(* Logix 5000 project; controller SX_V040001_C001 vendor 1 type 14 code 77 rev 16.23; software revision 16.04; part 3 of 35 *)
(* tags used below, declared in another part *)
   ALARM_BITS : INT[10];
   ALL_KINDS : INT[90];
   Basic : INT;
   G_DInput : DINT[3];
   G_DOutput : DINT[3];
   m_alarm_exist : BOOL;
   m_notstop : BOOL;
   METERING : INT[44];
   PARAMETER : INT[501];
   T_MET1_END : TIMER;
   T_MET2_END : TIMER;
   T_MET3_END : TIMER;
   T_MET4_END : TIMER;
   T_MET_VALVE_1 : TIMER;
   T_MET_VALVE_2 : TIMER;
   T_MET_VALVE_3 : TIMER;
   T_MET_VALVE_4 : TIMER;
   T_MET_VALVE_5 : TIMER;
   Z20 : COUNTER;
   Z21 : COUNTER;
   Z22 : COUNTER;
   Z23 : COUNTER;
   Z24 : COUNTER;
   Z25 : COUNTER;
   Z26 : COUNTER;
   Z27 : COUNTER;
   Z28 : COUNTER;
(* MainProgram, continued *)

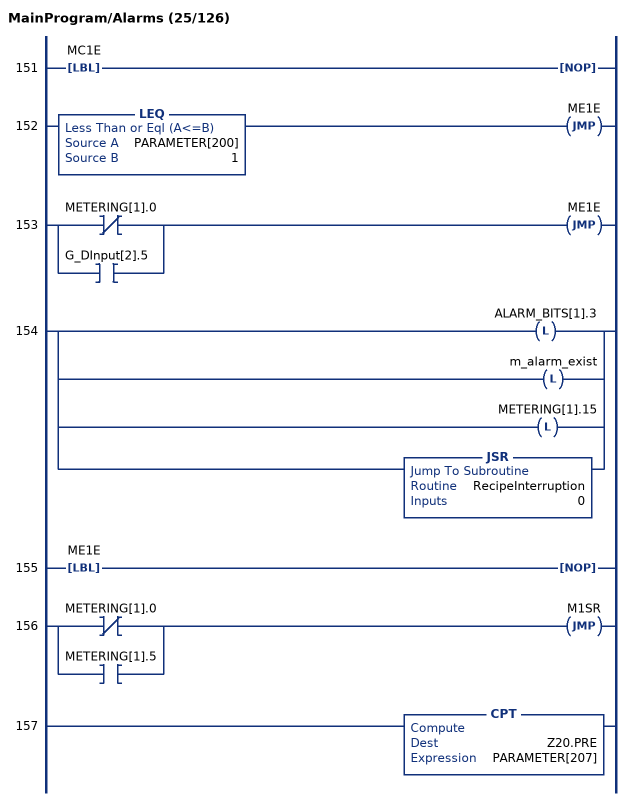
   [picture p46: MainProgram/Alarms rungs 151-157]
   151: LBL(MC1E)NOP();
   152: LEQ(PARAMETER[200],1)JMP(ME1E);
   153: [XIO(METERING[1].0) ,XIC(G_DInput[2].5) ]JMP(ME1E);
   154: [OTL(ALARM_BITS[1].3) ,OTL(m_alarm_exist) ,OTL(METERING[1].15) ,JSR(RecipeInterruption,0) ];
   155: LBL(ME1E)NOP();
   156: [XIO(METERING[1].0) ,XIC(METERING[1].5) ]JMP(M1SR);
   157: CPT(Z20.PRE,PARAMETER[207]);
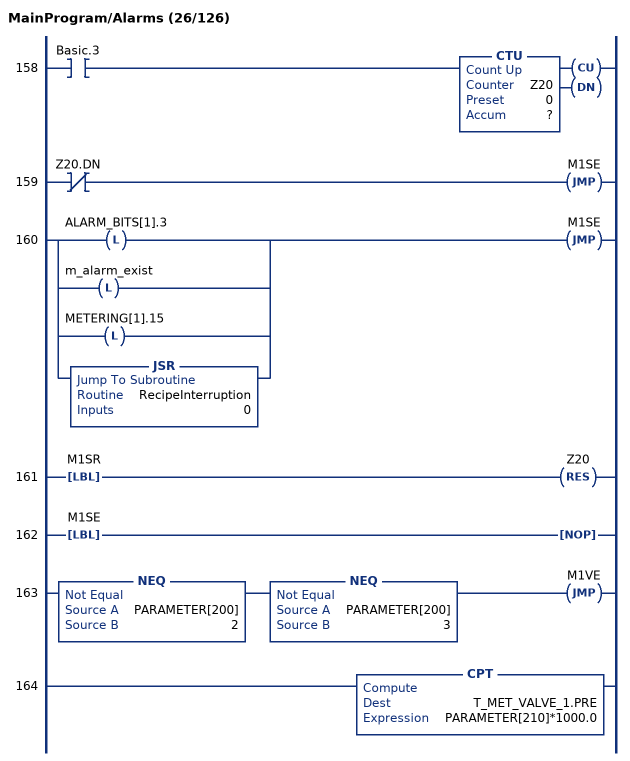
   158: XIC(Basic.3)CTU(Z20,?,?);
   159: XIO(Z20.DN)JMP(M1SE);
   160: [OTL(ALARM_BITS[1].3) ,OTL(m_alarm_exist) ,OTL(METERING[1].15) ,JSR(RecipeInterruption,0) ]JMP(M1SE);
   161: LBL(M1SR)RES(Z20);
   162: LBL(M1SE)NOP();
   163: NEQ(PARAMETER[200],2)NEQ(PARAMETER[200],3)JMP(M1VE);
   164: CPT(T_MET_VALVE_1.PRE,PARAMETER[210]*1000.0);
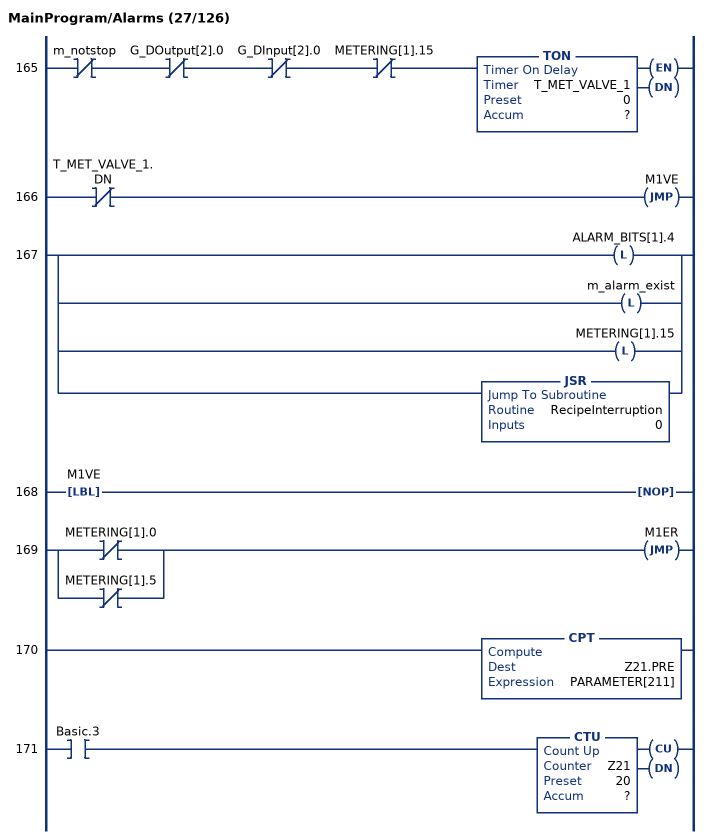
   165: XIO(m_notstop)XIO(G_DOutput[2].0)XIO(G_DInput[2].0)XIO(METERING[1].15)TON(T_MET_VALVE_1,?,?);
   166: XIO(T_MET_VALVE_1.DN)JMP(M1VE);
   167: [OTL(ALARM_BITS[1].4) ,OTL(m_alarm_exist) ,OTL(METERING[1].15) ,JSR(RecipeInterruption,0) ];
   168: LBL(M1VE)NOP();
   169: [XIO(METERING[1].0) ,XIO(METERING[1].5) ]JMP(M1ER);
   170: CPT(Z21.PRE,PARAMETER[211]);
   171: XIC(Basic.3)CTU(Z21,?,?);
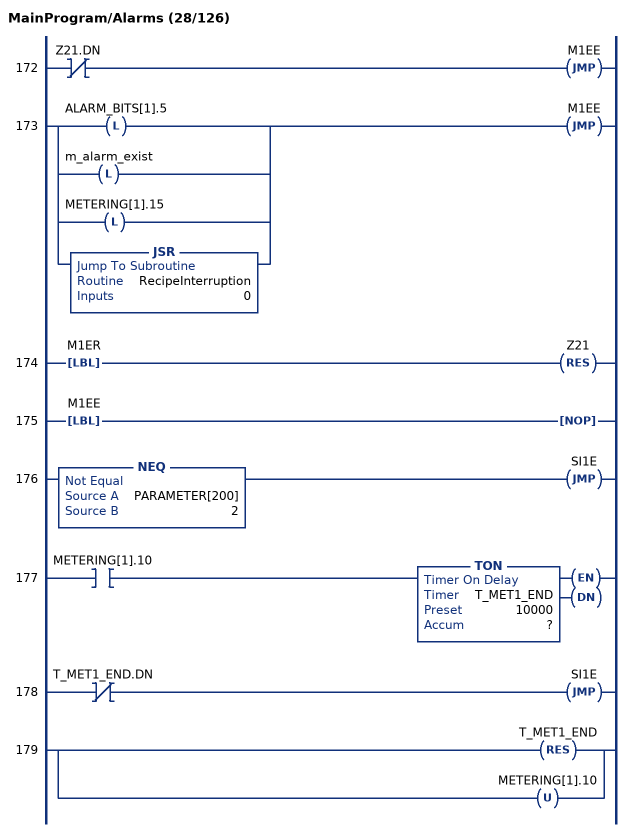
   172: XIO(Z21.DN)JMP(M1EE);
   173: [OTL(ALARM_BITS[1].5) ,OTL(m_alarm_exist) ,OTL(METERING[1].15) ,JSR(RecipeInterruption,0) ]JMP(M1EE);
   174: LBL(M1ER)RES(Z21);
   175: LBL(M1EE)NOP();
   176: NEQ(PARAMETER[200],2)JMP(SI1E);
   177: XIC(METERING[1].10)TON(T_MET1_END,?,?);
   178: XIO(T_MET1_END.DN)JMP(SI1E);
   179: [RES(T_MET1_END) ,OTU(METERING[1].10) ];
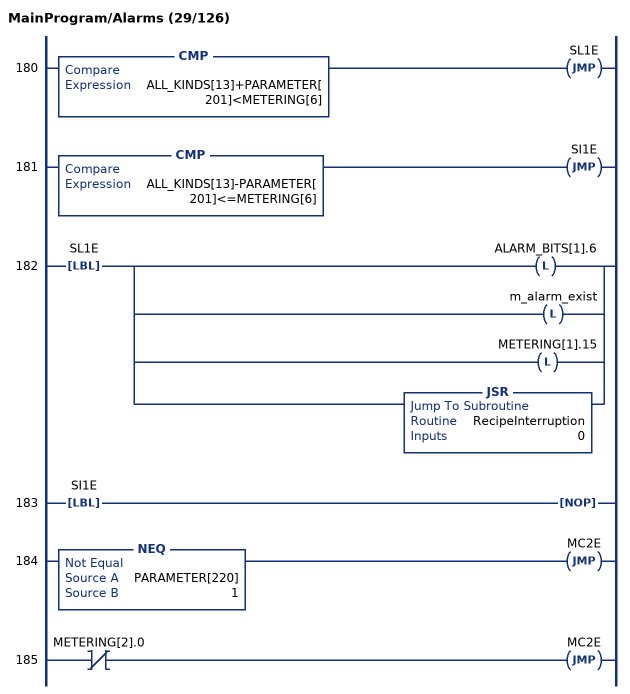
   180: CMP(ALL_KINDS[13]+PARAMETER[201]<METERING[6])JMP(SL1E);
   181: CMP(ALL_KINDS[13]-PARAMETER[201]<=METERING[6])JMP(SI1E);
   182: LBL(SL1E)[OTL(ALARM_BITS[1].6) ,OTL(m_alarm_exist) ,OTL(METERING[1].15) ,JSR(RecipeInterruption,0) ];
   183: LBL(SI1E)NOP();
   184: NEQ(PARAMETER[220],1)JMP(MC2E);
   185: XIO(METERING[2].0)JMP(MC2E);
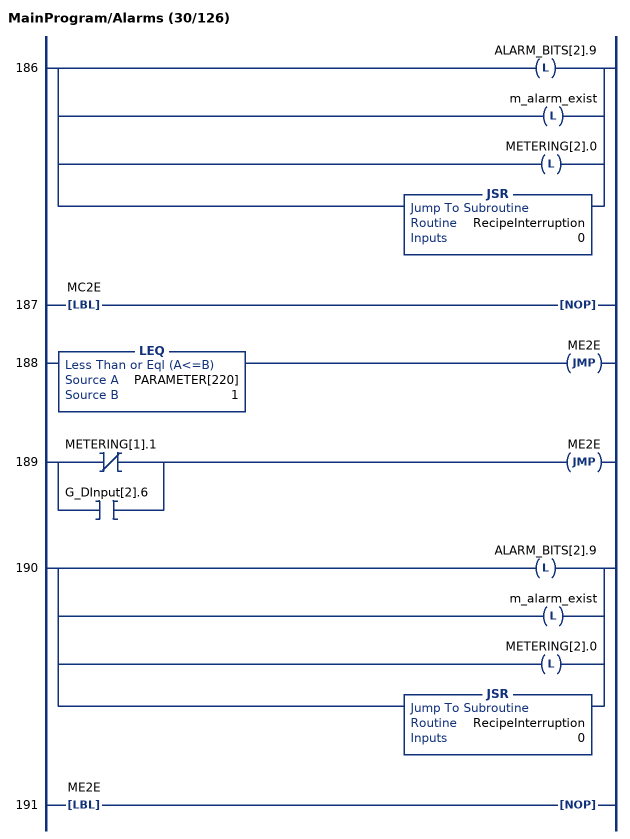
   186: [OTL(ALARM_BITS[2].9) ,OTL(m_alarm_exist) ,OTL(METERING[2].0) ,JSR(RecipeInterruption,0) ];
   187: LBL(MC2E)NOP();
   188: LEQ(PARAMETER[220],1)JMP(ME2E);
   189: [XIO(METERING[1].1) ,XIC(G_DInput[2].6) ]JMP(ME2E);
   190: [OTL(ALARM_BITS[2].9) ,OTL(m_alarm_exist) ,OTL(METERING[2].0) ,JSR(RecipeInterruption,0) ];
   191: LBL(ME2E)NOP();
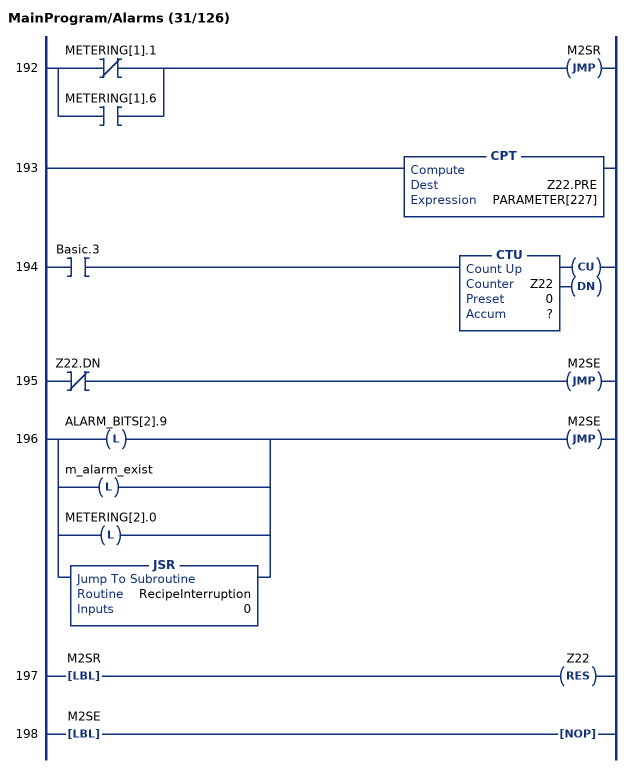
   192: [XIO(METERING[1].1) ,XIC(METERING[1].6) ]JMP(M2SR);
   193: CPT(Z22.PRE,PARAMETER[227]);
   194: XIC(Basic.3)CTU(Z22,?,?);
   195: XIO(Z22.DN)JMP(M2SE);
   196: [OTL(ALARM_BITS[2].9) ,OTL(m_alarm_exist) ,OTL(METERING[2].0) ,JSR(RecipeInterruption,0) ]JMP(M2SE);
   197: LBL(M2SR)RES(Z22);
   198: LBL(M2SE)NOP();
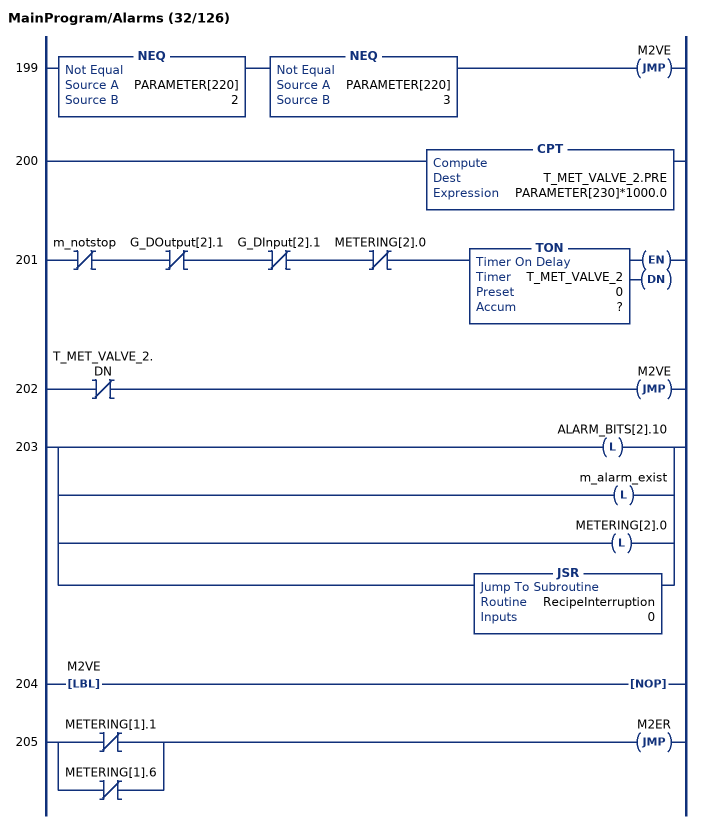
   199: NEQ(PARAMETER[220],2)NEQ(PARAMETER[220],3)JMP(M2VE);
   200: CPT(T_MET_VALVE_2.PRE,PARAMETER[230]*1000.0);
   201: XIO(m_notstop)XIO(G_DOutput[2].1)XIO(G_DInput[2].1)XIO(METERING[2].0)TON(T_MET_VALVE_2,?,?);
   202: XIO(T_MET_VALVE_2.DN)JMP(M2VE);
   203: [OTL(ALARM_BITS[2].10) ,OTL(m_alarm_exist) ,OTL(METERING[2].0) ,JSR(RecipeInterruption,0) ];
   204: LBL(M2VE)NOP();
   205: [XIO(METERING[1].1) ,XIO(METERING[1].6) ]JMP(M2ER);
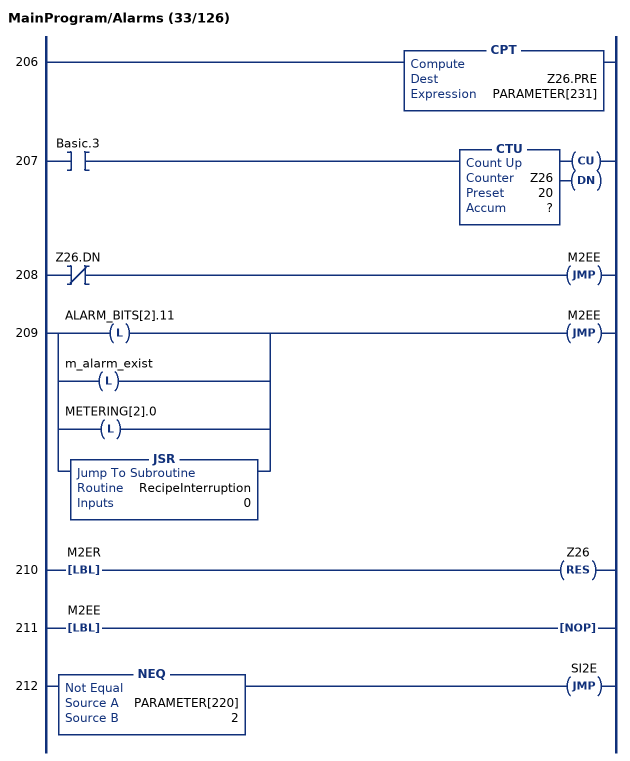
   206: CPT(Z26.PRE,PARAMETER[231]);
   207: XIC(Basic.3)CTU(Z26,?,?);
   208: XIO(Z26.DN)JMP(M2EE);
   209: [OTL(ALARM_BITS[2].11) ,OTL(m_alarm_exist) ,OTL(METERING[2].0) ,JSR(RecipeInterruption,0) ]JMP(M2EE);
   210: LBL(M2ER)RES(Z26);
   211: LBL(M2EE)NOP();
   212: NEQ(PARAMETER[220],2)JMP(SI2E);
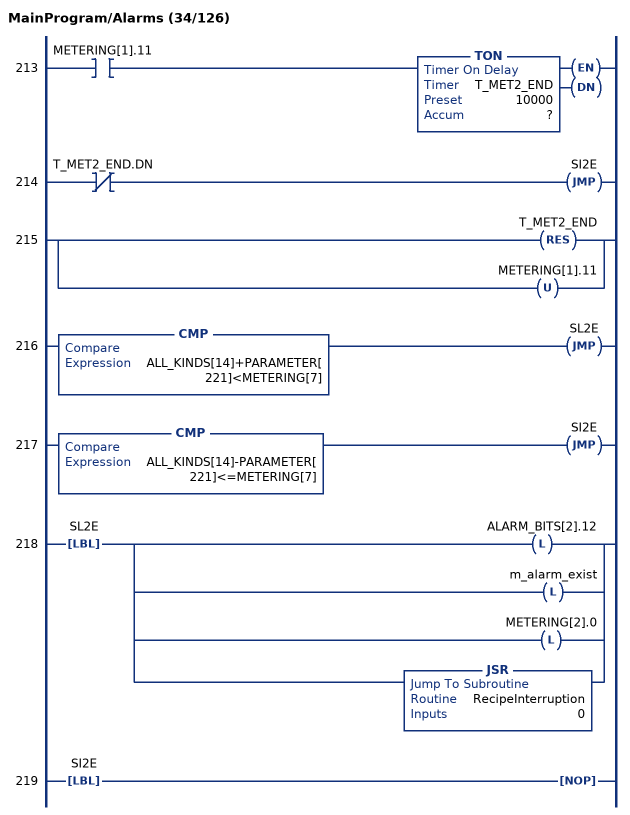
   213: XIC(METERING[1].11)TON(T_MET2_END,?,?);
   214: XIO(T_MET2_END.DN)JMP(SI2E);
   215: [RES(T_MET2_END) ,OTU(METERING[1].11) ];
   216: CMP(ALL_KINDS[14]+PARAMETER[221]<METERING[7])JMP(SL2E);
   217: CMP(ALL_KINDS[14]-PARAMETER[221]<=METERING[7])JMP(SI2E);
   218: LBL(SL2E)[OTL(ALARM_BITS[2].12) ,OTL(m_alarm_exist) ,OTL(METERING[2].0) ,JSR(RecipeInterruption,0) ];
   219: LBL(SI2E)NOP();
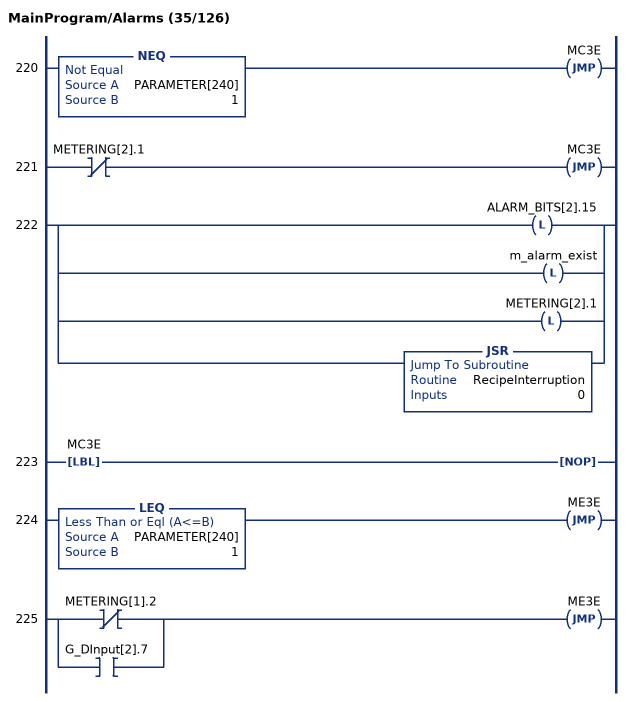
   220: NEQ(PARAMETER[240],1)JMP(MC3E);
   221: XIO(METERING[2].1)JMP(MC3E);
   222: [OTL(ALARM_BITS[2].15) ,OTL(m_alarm_exist) ,OTL(METERING[2].1) ,JSR(RecipeInterruption,0) ];
   223: LBL(MC3E)NOP();
   224: LEQ(PARAMETER[240],1)JMP(ME3E);
   225: [XIO(METERING[1].2) ,XIC(G_DInput[2].7) ]JMP(ME3E);
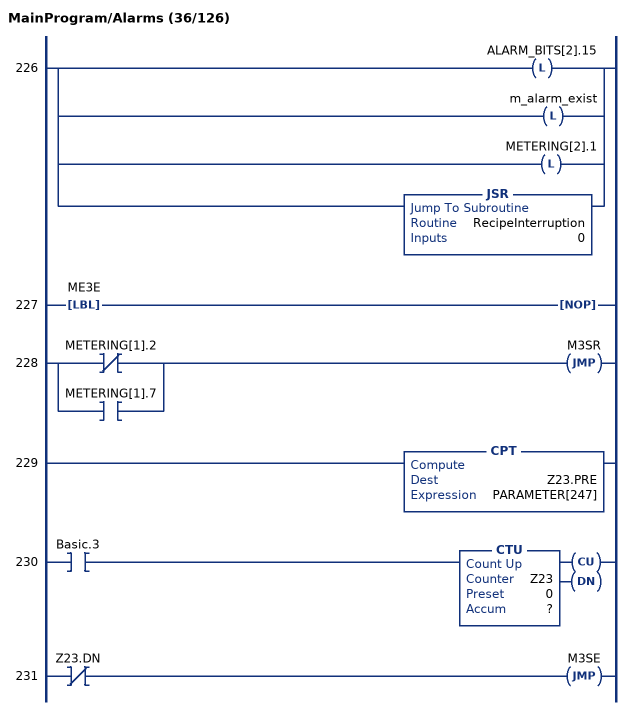
   226: [OTL(ALARM_BITS[2].15) ,OTL(m_alarm_exist) ,OTL(METERING[2].1) ,JSR(RecipeInterruption,0) ];
   227: LBL(ME3E)NOP();
   228: [XIO(METERING[1].2) ,XIC(METERING[1].7) ]JMP(M3SR);
   229: CPT(Z23.PRE,PARAMETER[247]);
   230: XIC(Basic.3)CTU(Z23,?,?);
   231: XIO(Z23.DN)JMP(M3SE);
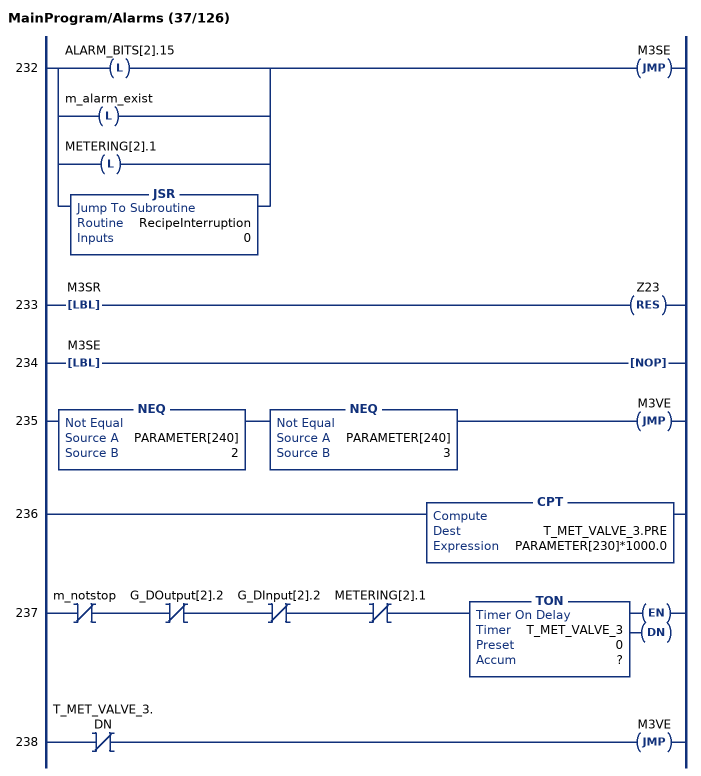
   232: [OTL(ALARM_BITS[2].15) ,OTL(m_alarm_exist) ,OTL(METERING[2].1) ,JSR(RecipeInterruption,0) ]JMP(M3SE);
   233: LBL(M3SR)RES(Z23);
   234: LBL(M3SE)NOP();
   235: NEQ(PARAMETER[240],2)NEQ(PARAMETER[240],3)JMP(M3VE);
   236: CPT(T_MET_VALVE_3.PRE,PARAMETER[230]*1000.0);
   237: XIO(m_notstop)XIO(G_DOutput[2].2)XIO(G_DInput[2].2)XIO(METERING[2].1)TON(T_MET_VALVE_3,?,?);
   238: XIO(T_MET_VALVE_3.DN)JMP(M3VE);
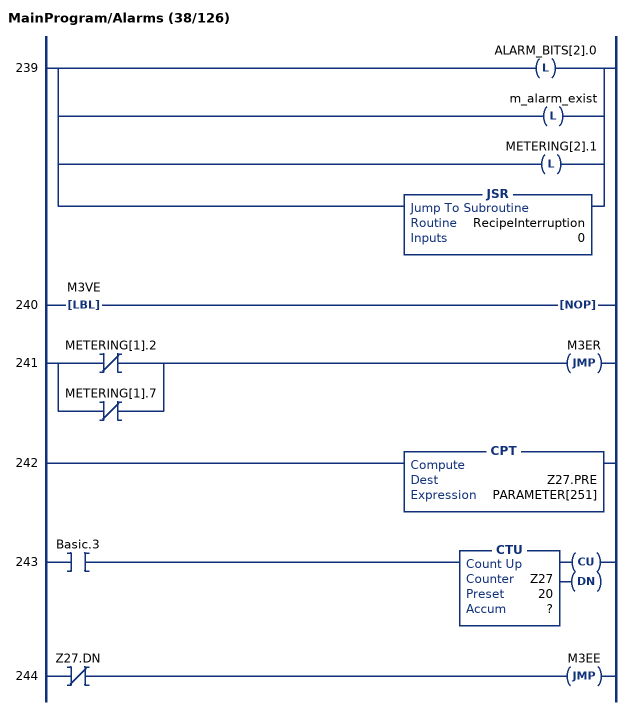
   239: [OTL(ALARM_BITS[2].0) ,OTL(m_alarm_exist) ,OTL(METERING[2].1) ,JSR(RecipeInterruption,0) ];
   240: LBL(M3VE)NOP();
   241: [XIO(METERING[1].2) ,XIO(METERING[1].7) ]JMP(M3ER);
   242: CPT(Z27.PRE,PARAMETER[251]);
   243: XIC(Basic.3)CTU(Z27,?,?);
   244: XIO(Z27.DN)JMP(M3EE);
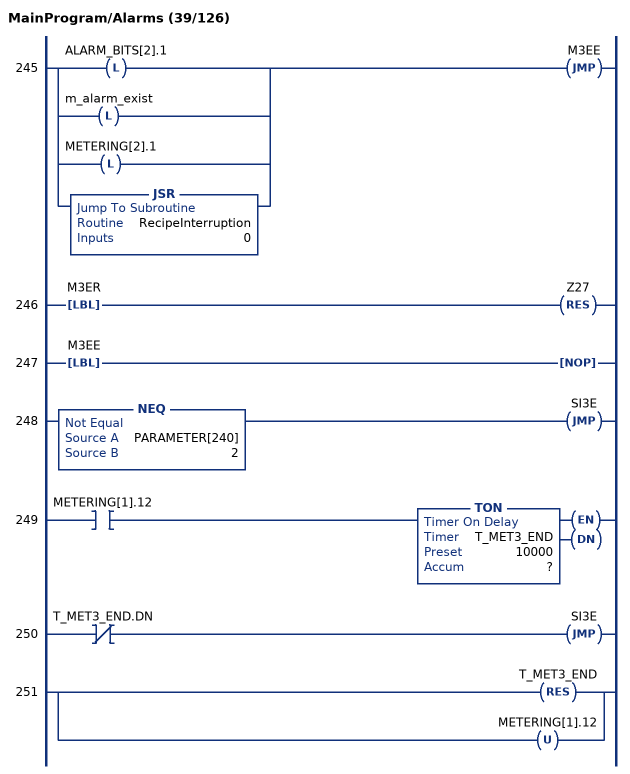
   245: [OTL(ALARM_BITS[2].1) ,OTL(m_alarm_exist) ,OTL(METERING[2].1) ,JSR(RecipeInterruption,0) ]JMP(M3EE);
   246: LBL(M3ER)RES(Z27);
   247: LBL(M3EE)NOP();
   248: NEQ(PARAMETER[240],2)JMP(SI3E);
   249: XIC(METERING[1].12)TON(T_MET3_END,?,?);
   250: XIO(T_MET3_END.DN)JMP(SI3E);
   251: [RES(T_MET3_END) ,OTU(METERING[1].12) ];
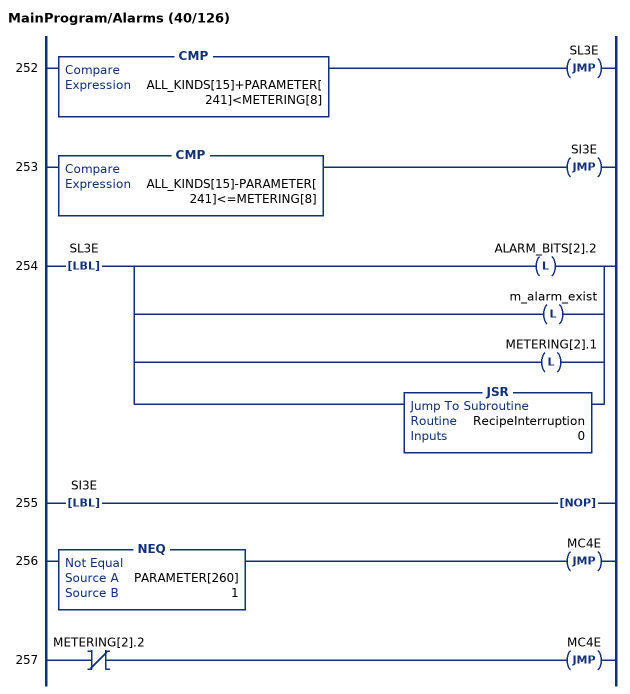
   252: CMP(ALL_KINDS[15]+PARAMETER[241]<METERING[8])JMP(SL3E);
   253: CMP(ALL_KINDS[15]-PARAMETER[241]<=METERING[8])JMP(SI3E);
   254: LBL(SL3E)[OTL(ALARM_BITS[2].2) ,OTL(m_alarm_exist) ,OTL(METERING[2].1) ,JSR(RecipeInterruption,0) ];
   255: LBL(SI3E)NOP();
   256: NEQ(PARAMETER[260],1)JMP(MC4E);
   257: XIO(METERING[2].2)JMP(MC4E);
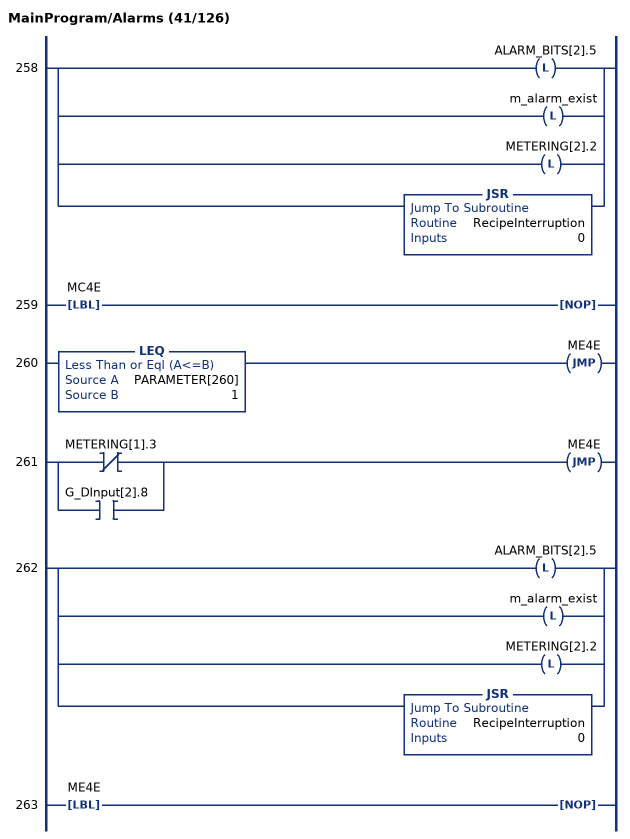
   258: [OTL(ALARM_BITS[2].5) ,OTL(m_alarm_exist) ,OTL(METERING[2].2) ,JSR(RecipeInterruption,0) ];
   259: LBL(MC4E)NOP();
   260: LEQ(PARAMETER[260],1)JMP(ME4E);
   261: [XIO(METERING[1].3) ,XIC(G_DInput[2].8) ]JMP(ME4E);
   262: [OTL(ALARM_BITS[2].5) ,OTL(m_alarm_exist) ,OTL(METERING[2].2) ,JSR(RecipeInterruption,0) ];
   263: LBL(ME4E)NOP();
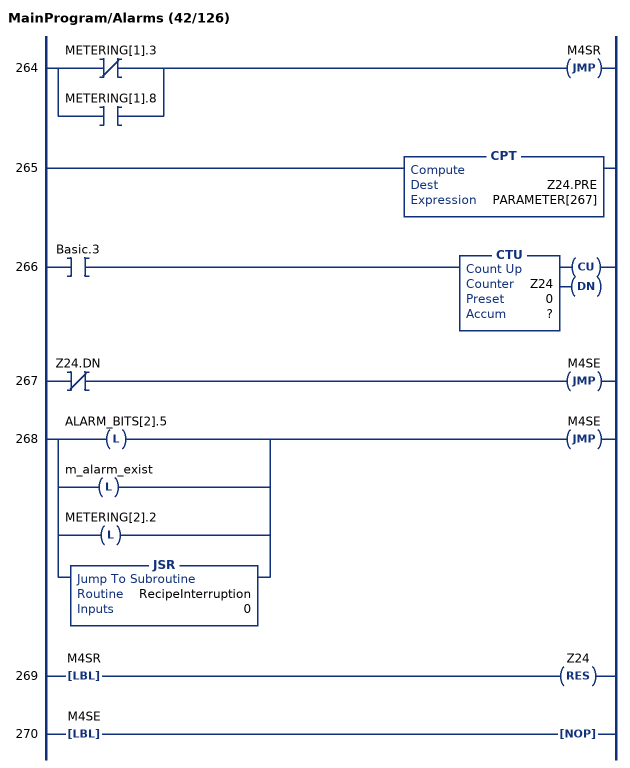
   264: [XIO(METERING[1].3) ,XIC(METERING[1].8) ]JMP(M4SR);
   265: CPT(Z24.PRE,PARAMETER[267]);
   266: XIC(Basic.3)CTU(Z24,?,?);
   267: XIO(Z24.DN)JMP(M4SE);
   268: [OTL(ALARM_BITS[2].5) ,OTL(m_alarm_exist) ,OTL(METERING[2].2) ,JSR(RecipeInterruption,0) ]JMP(M4SE);
   269: LBL(M4SR)RES(Z24);
   270: LBL(M4SE)NOP();
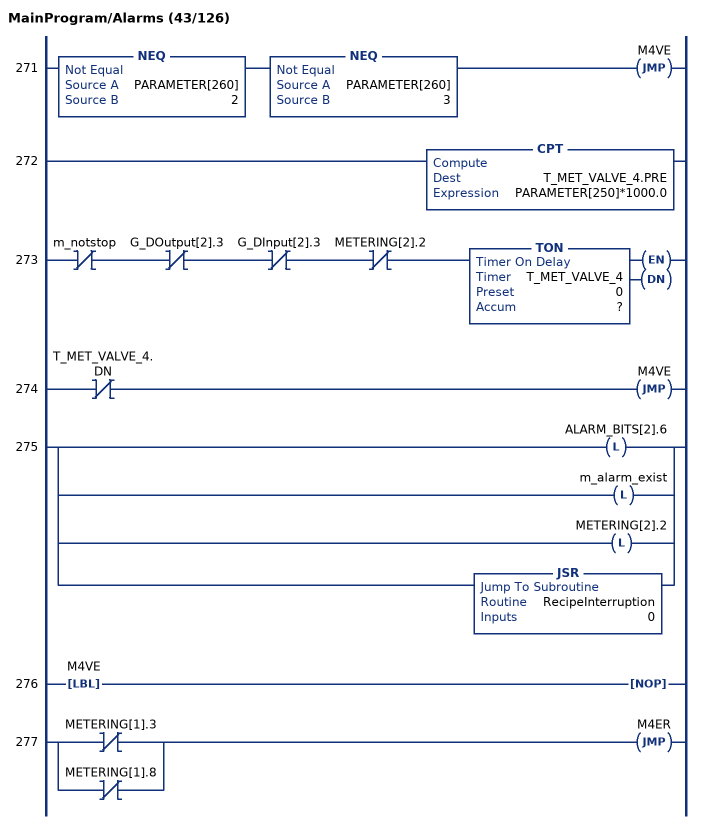
   271: NEQ(PARAMETER[260],2)NEQ(PARAMETER[260],3)JMP(M4VE);
   272: CPT(T_MET_VALVE_4.PRE,PARAMETER[250]*1000.0);
   273: XIO(m_notstop)XIO(G_DOutput[2].3)XIO(G_DInput[2].3)XIO(METERING[2].2)TON(T_MET_VALVE_4,?,?);
   274: XIO(T_MET_VALVE_4.DN)JMP(M4VE);
   275: [OTL(ALARM_BITS[2].6) ,OTL(m_alarm_exist) ,OTL(METERING[2].2) ,JSR(RecipeInterruption,0) ];
   276: LBL(M4VE)NOP();
   277: [XIO(METERING[1].3) ,XIO(METERING[1].8) ]JMP(M4ER);
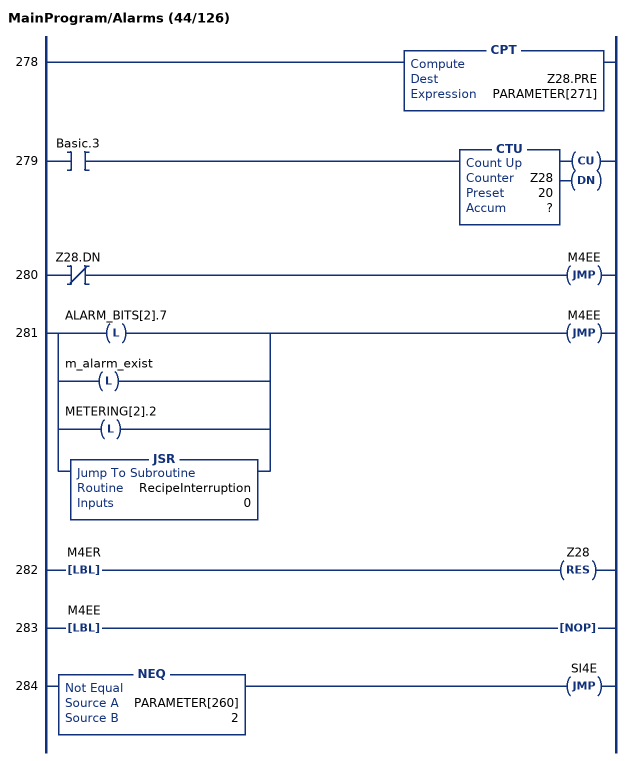
   278: CPT(Z28.PRE,PARAMETER[271]);
   279: XIC(Basic.3)CTU(Z28,?,?);
   280: XIO(Z28.DN)JMP(M4EE);
   281: [OTL(ALARM_BITS[2].7) ,OTL(m_alarm_exist) ,OTL(METERING[2].2) ,JSR(RecipeInterruption,0) ]JMP(M4EE);
   282: LBL(M4ER)RES(Z28);
   283: LBL(M4EE)NOP();
   284: NEQ(PARAMETER[260],2)JMP(SI4E);
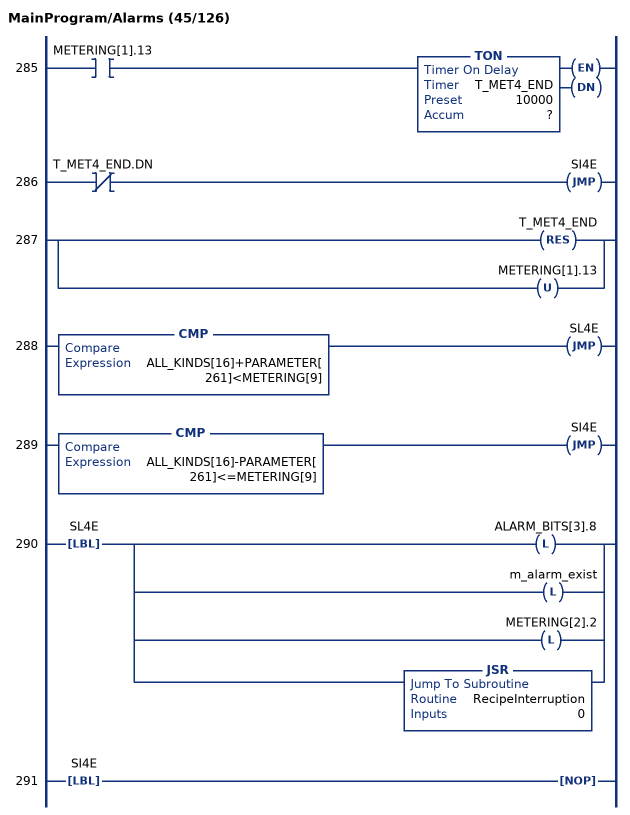
   285: XIC(METERING[1].13)TON(T_MET4_END,?,?);
   286: XIO(T_MET4_END.DN)JMP(SI4E);
   287: [RES(T_MET4_END) ,OTU(METERING[1].13) ];
   288: CMP(ALL_KINDS[16]+PARAMETER[261]<METERING[9])JMP(SL4E);
   289: CMP(ALL_KINDS[16]-PARAMETER[261]<=METERING[9])JMP(SI4E);
   290: LBL(SL4E)[OTL(ALARM_BITS[3].8) ,OTL(m_alarm_exist) ,OTL(METERING[2].2) ,JSR(RecipeInterruption,0) ];
   291: LBL(SI4E)NOP();
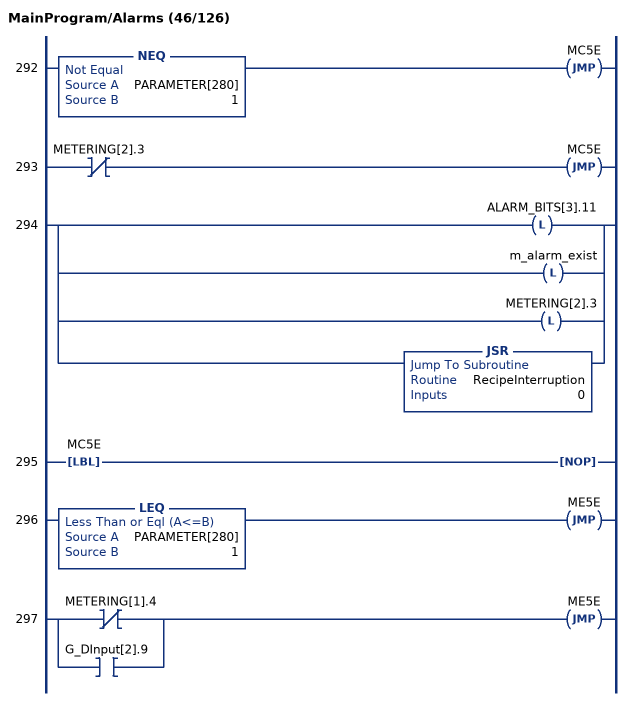
   292: NEQ(PARAMETER[280],1)JMP(MC5E);
   293: XIO(METERING[2].3)JMP(MC5E);
   294: [OTL(ALARM_BITS[3].11) ,OTL(m_alarm_exist) ,OTL(METERING[2].3) ,JSR(RecipeInterruption,0) ];
   295: LBL(MC5E)NOP();
   296: LEQ(PARAMETER[280],1)JMP(ME5E);
   297: [XIO(METERING[1].4) ,XIC(G_DInput[2].9) ]JMP(ME5E);
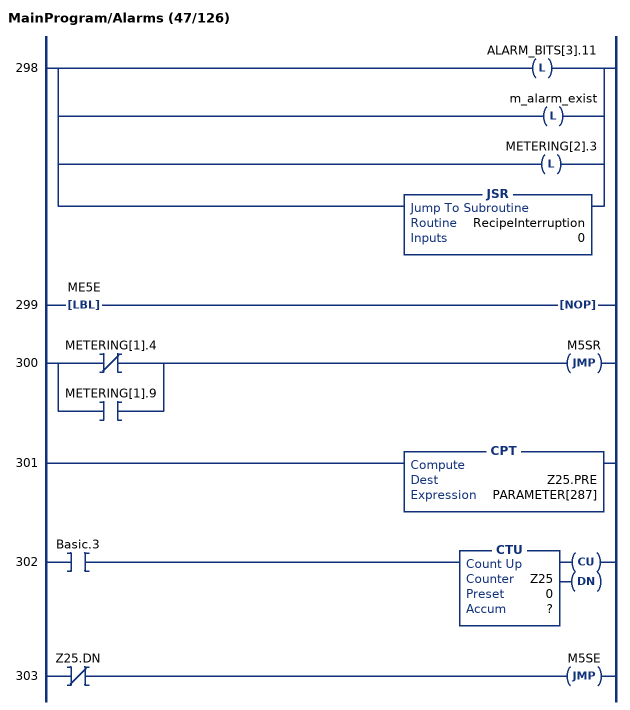
   298: [OTL(ALARM_BITS[3].11) ,OTL(m_alarm_exist) ,OTL(METERING[2].3) ,JSR(RecipeInterruption,0) ];
   299: LBL(ME5E)NOP();
   300: [XIO(METERING[1].4) ,XIC(METERING[1].9) ]JMP(M5SR);
   301: CPT(Z25.PRE,PARAMETER[287]);
   302: XIC(Basic.3)CTU(Z25,?,?);
   303: XIO(Z25.DN)JMP(M5SE);
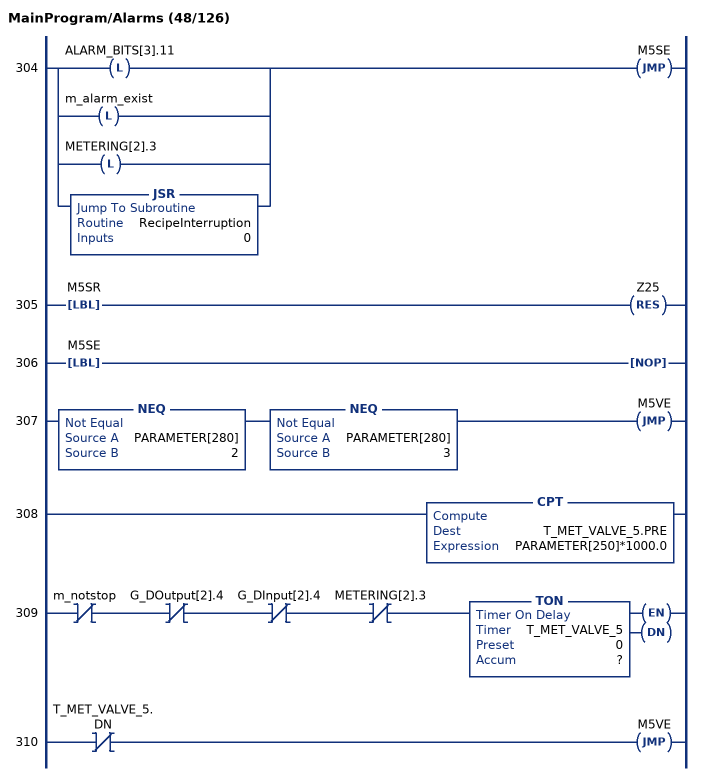
   304: [OTL(ALARM_BITS[3].11) ,OTL(m_alarm_exist) ,OTL(METERING[2].3) ,JSR(RecipeInterruption,0) ]JMP(M5SE);
   305: LBL(M5SR)RES(Z25);
   306: LBL(M5SE)NOP();
   307: NEQ(PARAMETER[280],2)NEQ(PARAMETER[280],3)JMP(M5VE);
   308: CPT(T_MET_VALVE_5.PRE,PARAMETER[250]*1000.0);
   309: XIO(m_notstop)XIO(G_DOutput[2].4)XIO(G_DInput[2].4)XIO(METERING[2].3)TON(T_MET_VALVE_5,?,?);
   310: XIO(T_MET_VALVE_5.DN)JMP(M5VE);
